Staubli VAL3: USPY.pgx

public program uSpy()
  local num lKey
begin
  do
    lKey=workingMode()
    if lKey==4
      userPage(false)
    endIf
    delay(0)
    delay(0)
  until false
end
